# EPICS autosave request: opticsApp/Db/flexCombinedMotion_settings.req
file motor_settings.req P=$(P),M=$(M)

$(P)$(M):mode.VAL
$(P)$(M):setPoint.VAL
$(P)$(M):setPoint.EGU
$(P)$(M):setPoint.DESC
$(P)$(M):setPoint.PREC
$(P)$(M):deadband.VAL
$(P)$(M):deadband.PREC
$(P)$(M):upperLimit.VAL
$(P)$(M):upperLimit.PREC
$(P)$(M):homePos.VAL
$(P)$(M):homePos.PREC
$(P)$(M):lowerLimit.VAL
$(P)$(M):lowerLimit.PREC
